// Sensors signal simulation
FUNCTION_BLOCK FB_SensorsSimulation
VAR_INPUT
	bEnable: BOOL;								// Enable sensor simulation
	 
	bRotateTable: BOOL;							// Signal to run the rotating table motor
	bLinearSliderMoveToPick : BOOL;     		// Signal to move the slider to the picking position
	bLinearSliderMoveToPlace : BOOL;    		// Signal to move the slider to the placing position
	
	tPartSensorDelay: TIME;						// Delay before the part sensor signal simulation
	tLinearSliderPickPosSensorDelay : TIME;		// Delay before the linear slider picking position sensor signal simulation
	tLinearSliderPlacePosSensorDelay : TIME;	// Delay before the linear slider placing position sensor signal simulation
	
	tStrobeDuration :TIME := T#1S;				// Duration of the simulated sensor signals
END_VAR
VAR_OUTPUT
	bPartSensorSignal: BOOL; 					// Simulated part sensor signal
	bLinearSliderPickPosSensorSignal: BOOL;		// Simulated linear slider picking position sensor
	bLinearSliderPlacePosSensorSignal: BOOL;	// Simulated linear slider placing position sensor
END_VAR
VAR
	fbPartSensorDelayTmr: TON;					// Part sensor delay timer
	fbPartSensorStrobeTmr: TP;					// Simulated part sensor signal strobe
	
	fbLinearSliderPickPosSensorDelayTmr: TON;	// Linear slider picking position sensor delay timer
	fbLinearSliderPlacePosSensorDelayTmr: TON;	// Simulated linear slider placing position sensor strobe
	
	
	fbLinearSliderPickPosSensorStrobeTmr: TP;	// Linear slider placing position sensor delay timer
	fbLinearSliderPlacePosSensorStrobeTmr: TP;	// Simulated linear slider picking position sensor strobe
	
				
END_VAR

{region "Part sensor simulation"}
fbPartSensorDelayTmr(IN:= bEnable AND bRotateTable, 
					 PT:= tPartSensorDelay, 
					 Q=> , 
 					 ET=> );
fbPartSensorStrobeTmr(IN:= fbPartSensorDelayTmr.Q, 
					  PT:= tStrobeDuration, 
					  Q=> bPartSensorSignal, 
					  ET=> );
{endregion}						 

{region "Slider pick position sensor"}					
fbLinearSliderPickPosSensorDelayTmr(IN:= bEnable AND bLinearSliderMoveToPick, 
									PT:= tLinearSliderPickPosSensorDelay, 
									Q=> , 
									ET=> );
fbLinearSliderPickPosSensorStrobeTmr(IN:= fbLinearSliderPickPosSensorDelayTmr.Q, 
									PT:= tStrobeDuration, 
									Q=> bLinearSliderPickPosSensorSignal, 
									ET=> );
{endregion}										 

{region "Slider place position sensor"}										
fbLinearSliderPlacePosSensorDelayTmr(IN:= bEnable AND bLinearSliderMoveToPlace, 
									PT:= tLinearSliderPlacePosSensorDelay, 
									Q=> , 
									ET=> );
fbLinearSliderPlacePosSensorStrobeTmr(IN:= fbLinearSliderPlacePosSensorDelayTmr.Q, 
									PT:= tStrobeDuration, 
									Q=> bLinearSliderPlacePosSensorSignal, 
									ET=> );
{endregion}

END_FUNCTION_BLOCK

(* stored: Version 1.1.0.1, ProductVersion 3.1.4024.12
   POU FB_SensorsSimulation: Id {d0951dc2-7fe7-4eb0-9a9c-218b7ed9d559}, SpecialFunc None *)
